DATA_BLOCK "DB2005_SD"
TITLE = DB2005_SD
{ S7_Optimized_Access := 'FALSE' }
AUTHOR : ABH
FAMILY : ZeusControl
VERSION : 1.0
//Bloque de datos salida digital
   STRUCT
      SD : Array[0.."N_MAX_DISP_SD"] of "UDT_ZC_DISP_SD";
      Mux { S7_SetPoint := 'False'} : Array[0.."N_MAX_MUX_DISP"] of "UDT_ZC_DISP_MUX_SD";
      Agrup : Array[0.."N_MAX_DISP_AGRUP"] of "UDT_ZC_DISP_AGRUP";
   END_STRUCT;


BEGIN
   SD[0].Hmi_Estado := 0;
   SD[0].Estado_AutoMan := FALSE;
   SD[0].Estado_Activado := FALSE;
   SD[0].Estado_Enclavado := FALSE;
   SD[0].Orden_ActivarManual := FALSE;
   SD[0].Orden_ActivarAuto := FALSE;
   SD[0].Config_Habilitar := FALSE;
   SD[0].Config_HabilitarRetardoAct := FALSE;
   SD[0].Config_HabilitarRetardoDes := FALSE;
   SD[0].Config_HabilitarInvertir := FALSE;
   SD[0].Aux_oldActivado := FALSE;
   SD[0].Aux_oldAutoMan := FALSE;
   SD[0].Estado_SeguridadOk := TRUE;
   SD[0].Config_GrupoAlarma := 0;
   SD[0].Config_DireccionSalidaByte := 0;
   SD[0].Config_DireccionSalidaBit := 0;
   SD[0].Tiempos_SetPointTiempoAct := 3;
   SD[0].Tiempos_SetPointTiempoDes := 3;
   SD[0].Tiempos_TiempoAct := 0;
   SD[0].Tiempos_TiempoDes := 0;
   SD[1].Hmi_Estado := 10;
   SD[1].Estado_AutoMan := TRUE;
   SD[1].Estado_Activado := TRUE;
   SD[1].Estado_Enclavado := FALSE;
   SD[1].Orden_ActivarManual := TRUE;
   SD[1].Orden_ActivarAuto := FALSE;
   SD[1].Config_Habilitar := FALSE;
   SD[1].Config_HabilitarRetardoAct := FALSE;
   SD[1].Config_HabilitarRetardoDes := FALSE;
   SD[1].Config_HabilitarInvertir := FALSE;
   SD[1].Aux_oldActivado := FALSE;
   SD[1].Aux_oldAutoMan := TRUE;
   SD[1].Estado_SeguridadOk := TRUE;
   SD[1].Config_GrupoAlarma := 0;
   SD[1].Config_DireccionSalidaByte := 101;
   SD[1].Config_DireccionSalidaBit := 5;
   SD[1].Tiempos_SetPointTiempoAct := 3;
   SD[1].Tiempos_SetPointTiempoDes := 3;
   SD[1].Tiempos_TiempoAct := 0;
   SD[1].Tiempos_TiempoDes := 0;
   Mux[0].Habilitar := TRUE;
   Mux[0].ExisteCambio := FALSE;
   Mux[0].MaxVisible := FALSE;
   Mux[0].Index := 0;
   Mux[0].oldIndex := 0;
   Mux[0].SD.Hmi_Estado := 0;
   Mux[0].SD.Estado_AutoMan := FALSE;
   Mux[0].SD.Estado_Activado := FALSE;
   Mux[0].SD.Estado_Enclavado := FALSE;
   Mux[0].SD.Orden_ActivarManual := FALSE;
   Mux[0].SD.Orden_ActivarAuto := FALSE;
   Mux[0].SD.Config_Habilitar := FALSE;
   Mux[0].SD.Config_HabilitarRetardoAct := FALSE;
   Mux[0].SD.Config_HabilitarRetardoDes := FALSE;
   Mux[0].SD.Config_HabilitarInvertir := FALSE;
   Mux[0].SD.Aux_oldActivado := FALSE;
   Mux[0].SD.Aux_oldAutoMan := FALSE;
   Mux[0].SD.Estado_SeguridadOk := TRUE;
   Mux[0].SD.Config_GrupoAlarma := 0;
   Mux[0].SD.Config_DireccionSalidaByte := 0;
   Mux[0].SD.Config_DireccionSalidaBit := 0;
   Mux[0].SD.Tiempos_SetPointTiempoAct := 3;
   Mux[0].SD.Tiempos_SetPointTiempoDes := 3;
   Mux[0].SD.Tiempos_TiempoAct := 0;
   Mux[0].SD.Tiempos_TiempoDes := 0;
   Mux[1].Habilitar := TRUE;
   Mux[1].ExisteCambio := FALSE;
   Mux[1].MaxVisible := FALSE;
   Mux[1].Index := 0;
   Mux[1].oldIndex := 0;
   Mux[1].SD.Hmi_Estado := 0;
   Mux[1].SD.Estado_AutoMan := FALSE;
   Mux[1].SD.Estado_Activado := FALSE;
   Mux[1].SD.Estado_Enclavado := FALSE;
   Mux[1].SD.Orden_ActivarManual := FALSE;
   Mux[1].SD.Orden_ActivarAuto := FALSE;
   Mux[1].SD.Config_Habilitar := FALSE;
   Mux[1].SD.Config_HabilitarRetardoAct := FALSE;
   Mux[1].SD.Config_HabilitarRetardoDes := FALSE;
   Mux[1].SD.Config_HabilitarInvertir := FALSE;
   Mux[1].SD.Aux_oldActivado := FALSE;
   Mux[1].SD.Aux_oldAutoMan := FALSE;
   Mux[1].SD.Estado_SeguridadOk := TRUE;
   Mux[1].SD.Config_GrupoAlarma := 0;
   Mux[1].SD.Config_DireccionSalidaByte := 0;
   Mux[1].SD.Config_DireccionSalidaBit := 0;
   Mux[1].SD.Tiempos_SetPointTiempoAct := 3;
   Mux[1].SD.Tiempos_SetPointTiempoDes := 3;
   Mux[1].SD.Tiempos_TiempoAct := 0;
   Mux[1].SD.Tiempos_TiempoDes := 0;
   Agrup[0].AlgunaEnManual := FALSE;
   Agrup[0].AlgunaAlarma := FALSE;
   Agrup[0].NuevaAlarma := FALSE;
   Agrup[1].AlgunaEnManual := FALSE;
   Agrup[1].AlgunaAlarma := FALSE;
   Agrup[1].NuevaAlarma := FALSE;

END_DATA_BLOCK

